FUNCTION_BLOCK CiA_DS402Statusword_Parker EXTENDS CiA_DS402Statusword
VAR_INPUT
END_VAR
VAR_OUTPUT	
	TargetReached				: BOOL; // Bit 10 
	Running						: BOOL; //Bit 14
END_VAR

METHOD PUBLIC readStatusword : BOOL
VAR_INPUT
	Statusword 					:	UINT;
END_VAR


	TargetReached											:= Statusword.10;
	Running													:= Statusword.14;

	readStatusword											:= SUPER^.readStatusword(Statusword);
END_METHOD

END_FUNCTION_BLOCK

(* stored: Version 1.1.0.1, ProductVersion 3.1.4024.3
   POU CiA_DS402Statusword_Parker: Id {450a9c00-11ee-4927-98b5-e9c717d81103}, SpecialFunc None
   Method readStatusword: Id {951a9c3f-4c82-480b-a468-f35954274f7b} *)
